Staubli VAL3: onRun.pgx

public program onRun(string& x_sItem[])
  local num l_nValue
  local num l_nVelocity
begin
  //
  // convert to a num

  bAxisMove=true
  aioSet(io:MbAO_b8Axis,1)
  aioSet(io:MbAO_bMoveToPos,0)
  toNum(x_sItem,l_nValue,true)
  // NB the robot will no STOP
//  aioSet(io:MbAI_bAxis8Reac,0)
  delay(0.5)
  l_nVelocity=speedScale()
  l_nVelocity=700*l_nVelocity/100
  l_nVelocity=round(l_nVelocity)
  l_nValue=round(l_nValue)
  aioSet(io:MbAO_aMovePosL8,0)
  aioSet(io:MbAO_aMovePosH8,2.554265*l_nValue)
  aioSet(io:MbAO_aMoveDis8,1)
  aioSet(io:MbAO_aVelocity8,l_nVelocity)
  aioSet(io:MbAO_bMovePos8,1)
  delay(0.5)
  wait(aioGet(io:MbAI_bAxis8Reac)==0)
  wait(aioGet(io:MbAI_bAxis8Reac)==1)
  aioSet(io:MbAO_bMovePos8,0)
  aioSet(io:MbAO_aMoveDis8,0)
  aioSet(io:MbAO_b8Axis,0)
  bAxisMove=false
end
